// TIA Portal V17 export
// export: Created 2025-03-07T09:17:35.1423807Z, ExportSetting WithDefaults, DisplayName Totally Integrated Automation Portal, DisplayVersion V17 Update 8, DisplayName TIA Portal Openness, DisplayVersion V17 Update 8, DisplayName TIA Portal Version Control Interface, DisplayVersion V17, DisplayName SINAMICS Startdrive Advanced, DisplayVersion V17 SP2, DisplayName SINAMICS Startdrive G110M, G120, G120C, G120D, G120P, G115D, DisplayVersion V17 SP2, DisplayName SINAMICS Startdrive G130, G150, S120, S150, SINAMICS MV, S210, DisplayVersion V17 SP2, DisplayName STEP 7 Professional, DisplayVersion V17 Update 8, DisplayName SINUMERIK ONE STEP 7 Toolbox, DisplayVersion V17 Update 12, DisplayName SINUMERIK 840D sl STEP 7 Toolbox, DisplayVersion V17 Update 12, DisplayName STEP 7 Safety, DisplayVersion V17 Update 6, DisplayName WinCC Advanced, DisplayVersion V17 Update 8
DATA_BLOCK "DB440_MACHINE_ALARM_DECODING"   // DB440
{ S7_Optimized_Access := 'FALSE'; DB_Accessible_From_OPC_UA := 'FALSE' }
AUTHOR : ETXETAR
VERSION : 1.0
// stored: AutoNumber false, DBAccessibleFromOPCUA false, DBAccessibleFromWebserver true, IsOnlyStoredInLoadMemory false, IsWriteProtectedInAS false
   VAR RETAIN
      GLOBAL_ALARMS_MACHINE { S7_SetPoint := 'True'} : "MACHINE ALARM";
      ALARMS_CENTRAL { S7_SetPoint := 'True'} : "UNIT ALARM";
      ALARMS_UNIT_01 : Struct
         GLOBAL : "UNIT ALARM";
         ST0_TRANSFER : "UNIT ALARM";
         ST1_LOAD_UNLOAD : "UNIT ALARM";
         ST2_SPARE : "UNIT ALARM";
         ST3_CLADDING : "UNIT ALARM";
         ST4_CLEANING : "UNIT ALARM";
         HOPPERS : "UNIT ALARM";
      END_STRUCT;
      ALARMS_UNIT_02 : Struct
         GLOBAL : "UNIT ALARM";
         ST0_TRANSFER : "UNIT ALARM";
         ST1_LOAD_UNLOAD : "UNIT ALARM";
         ST2_MEASURING : "UNIT ALARM";
         ST3_CLADDING : "UNIT ALARM";
         ST4_CLEANING : "UNIT ALARM";
         HOPPERS : "UNIT ALARM";
      END_STRUCT;
      ALARMS_UNIT_03 : "UNIT ALARM";
      ALARMS_UNIT_04 : "UNIT ALARM";
      PROGRAMMING_ALARM_DECODING : DInt;   // PROGRAMMING ALARM DECODING
      TIMER_ALARMS_DELAY { S7_SetPoint := 'True'} : TON_TIME;
   END_VAR
BEGIN
   TIMER_ALARMS_DELAY.PT := T#3s;
END_DATA_BLOCK
